{attribute 'pack_mode' := '1'}
TYPE ST_BINFILLER_MSG :
STRUCT
END_STRUCT
END_TYPE

(* stored: Version 1.1.0.1, ProductVersion 3.1.4024.12
   DUT ST_BINFILLER_MSG: Id {68ea041b-1075-40e3-bede-515b27c39237} *)
